FUNCTION_BLOCK SymbolPathStorage

VAR_OUTPUT
END_VAR
VAR_STAT
	aBoolInPaths : ARRAY[1..cMaxPaths] OF T_MaxString;
	aBoolOutPaths : ARRAY[1..cMaxPaths] OF T_MaxString;
	uiBoolInPathCtr : UINT := 1;
	uiBoolOutPathCtr : UINT := 1;
END_VAR
VAR CONSTANT
	cMaxPaths : UINT := 512;
END_VAR

END_FUNCTION_BLOCK

(* stored: Version 1.1.0.1, ProductVersion 3.1.4024.2
   POU SymbolPathStorage: Id {c0e9eca6-73c7-47b3-b528-a1392fd56dd4}, SpecialFunc None *)
